FUNCTION_BLOCK FB_MotionAxisDS402_TestDouble IMPLEMENTS I_MotionAxisDS402
VAR
    bError: BOOL;
    nErrorID: UDINT;
    sMessage : T_MAXSTRING;
    stMotionAxisStatus : ST_MotionAxisStatus;
    bConfigDone : BOOL;
END_VAR

METHOD AxisEnabled : BOOL
END_METHOD

(*
    Handle positive/negative backlash compensation
    User needs to set the direction of backlash from the sign of the compensation value
    Backlash compensation is disabled during referencing (homing).
    When direction is positive/negative, further movement in the negative/positive direction not compensated
    further movement in the negative/positive direction will be compensated
*)
METHOD BacklashCompensation
VAR_INPUT
    Enable	: BOOL := FALSE;
    RampVelo	: LREAL;
END_VAR
END_METHOD

PROPERTY ConfigDone : BOOL
GET
ConfigDone := bConfigDone;
END_GET
SET
bConfigDone := ConfigDone;
END_SET
END_PROPERTY

METHOD DisablePower
END_METHOD

METHOD DriveCommands
VAR_INPUT
    HomeCmd	: BOOL;
    NewMoveReq	: BOOL;
    EnableMode	: E_StageEnableMode;
END_VAR
END_METHOD

METHOD Halt
VAR_INPUT
    Deceleration	: LREAL := 0;
    Jerk	: LREAL := 0;
    BufferMode	: MC_BufferMode := MC_BufferMode.MC_Aborting;
END_VAR
END_METHOD

METHOD HaltDone
END_METHOD

METHOD Home
VAR_INPUT
    Position	: LREAL := .DEFAULT_HOME_POSITION;
    BufferMode	: MC_BufferMode;
END_VAR
END_METHOD

METHOD ModeConfigDone : BOOL
VAR_INPUT
    Mode	: E_EpicsMotorCmd;
END_VAR
 ModeConfigDone :=  bConfigDone;
END_METHOD

METHOD ModeOfOperation : BOOL
VAR_INPUT
    RecentModeOfOperation	: E_DS402OpMode;
END_VAR
END_METHOD

METHOD MoveAbsolute
VAR_INPUT
    Position	: LREAL;
    Velocity	: LREAL;
    Acceleration	: LREAL := 0;
    Deceleration	: LREAL := 0;
    Jerk	: LREAL := 0;
    BufferMode	: MC_BufferMode := MC_BufferMode.MC_Aborting;
END_VAR
END_METHOD

METHOD Power
VAR_INPUT
    Enable	: BOOL;
    Enable_Positive	: BOOL;
    Enable_Negative	: BOOL;
    Override	: LREAL;
    BufferMode	: MC_BufferMode;
END_VAR
END_METHOD

METHOD ReadAxisParams
VAR_INPUT
    Enable	: BOOL;
    RefreshDelay	: TIME;
END_VAR
END_METHOD

METHOD Reset
END_METHOD

METHOD ResetDone
END_METHOD

METHOD SaveAxisParams
VAR_INPUT
    Enable	: BOOL;
END_VAR
END_METHOD

PROPERTY Status : REFERENCE TO ST_MotionAxisStatus
GET
Status REF= stMotionAxisStatus;
END_GET
END_PROPERTY

END_FUNCTION_BLOCK

(* stored: Version 1.1.0.1
   POU FB_MotionAxisDS402_TestDouble: Id {77806d47-ac65-4da7-a599-d0f423642259}, SpecialFunc None
   Method AxisEnabled: Id {5ff88de4-575e-4374-aec8-16bb330a0f21}
   Method BacklashCompensation: Id {bf4738e3-e03f-4210-8d67-78a9614c3b23}
   Property ConfigDone: Id {293f2a35-f8b1-4e02-928d-6090a8d8fd2f}
   Get Get: Id {847a7378-c529-4f8f-8d37-c7b68dfff763}
   Set Set: Id {8e4bf5f7-f37c-45c4-a13a-97b537cb6c0e}
   Method DisablePower: Id {67d4c7d5-e408-429b-a2fc-f12a8f2f307b}
   Method DriveCommands: Id {4809421a-ad9b-4ec0-8380-a16bbba1e8bf}
   Method Halt: Id {24817d88-4d3a-4531-867f-0a5b18e50cb3}
   Method HaltDone: Id {6142ed56-20e6-4b7e-84d7-6bb060eaad96}
   Method Home: Id {2de1c4e2-757b-47b6-84b3-d845676f9de7}
   Method ModeConfigDone: Id {6077f8c2-be17-4f2f-80dd-8118e460311b}
   Method ModeOfOperation: Id {25325ca5-88b7-4b07-9393-8478c4f92c31}
   Method MoveAbsolute: Id {f7b91bdc-abd6-487d-ab94-c50c85da6522}
   Method Power: Id {1e779a14-4cae-4521-9b22-ad50ad5385f0}
   Method ReadAxisParams: Id {2d424ed8-d634-4f2e-8986-7cb9406ca020}
   Method Reset: Id {7cb8bf4f-c204-4086-b9cb-fb4943a5f116}
   Method ResetDone: Id {f1ca130c-0662-4c62-acfc-87bcc67bab0c}
   Method SaveAxisParams: Id {4650e62c-6837-41f8-8765-7a4b80e5af78}
   Property Status: Id {20cf4b89-8254-4cea-914b-f8629ff8572c}
   Get Get: Id {f5013c20-1dbd-4c70-820e-5e55d7d634b3} *)
